TYPE ST_LiftTable_Inp_OP :
STRUCT
	DriveUp				: BOOL; //Push button on Operator panel to drive lift up
	DriveDown			: BOOL; //Push button on Operator panel to drive lift down
	OPStartTransport	: BOOL; //Push button on Operator panel to set TU ready to move
END_STRUCT
END_TYPE

(* stored: Version 1.1.0.1, ProductVersion 3.1.4024.9
   DUT ST_LiftTable_Inp_OP: Id {cbaea96d-591c-46db-8b29-ce98e9739c8d} *)
